// TIA Portal V20 export
// export: Created 2025-12-01T14:57:01.9840998Z, ExportSetting None, DisplayName Totally Integrated Automation Portal, DisplayVersion V20 Update 3, DisplayName TIA Portal Openness, DisplayVersion V20 Update 3, DisplayName TIA Portal Version Control Interface, DisplayVersion V20 Update 3, DisplayName STEP 7 Professional, DisplayVersion V20 Update 3, DisplayName STEP 7 Safety, DisplayVersion V20 Update 2, DisplayName WinCC Basic/Comfort/Advanced, DisplayVersion V20 Update 3, DisplayName WinCC Professional, DisplayVersion V20 Update 3, DisplayName WinCC Unified, DisplayVersion V20 Update 3
FUNCTION "FC465_Elevador_Continuo_Building" : Void   // FC465, LAD
TITLE = ELEVADOR CONTINUO
{ S7_Optimized_Access := 'FALSE' }
VERSION : 1.0
// Control para un elevador continuo con una única entrada y una única salida. si requiere de más salidas es necesario aplicar otro control para el movimiento y para el transportador abatible
// stored: AutoNumber false, SetENOAutomatically false
   VAR_INPUT
      NumeroMesa : UInt;
      NumeroMesaEntrada : UInt;
      NumeroMesaSalida : UInt;
      Termico_TEnt : Bool;
      Termico_TSal : Bool;
      Termico_Elev : Bool;
      pHs_Ent : Bool;
      Prot_Ent : Bool;
      pHs_Sal : Bool;
      Prot_Sal : Bool;
      Det_Sincr_Entrada : Bool;
      Det_Salida_Paro : Bool;
      Det_Salida_Emerg : Bool;
      AVTF_Ant : Bool;
      PTF_Sig : Bool;
      V_Permiso_Entrada : UDInt;
      V_Presencia_Entrada : UDInt;
      V_Paro_Elev : UDInt;
      V_Paro_Sal_ms : UDInt;
   END_VAR
   VAR_IN_OUT
      MAux_FP_Sincr : Bool;
      MAux_FN_Entrada : Bool;
      MAux_FP_Salida : Bool;
      Mem_TmpParoSal : Bool;
      Mem_Paro_Elev : Bool;
      out_Elevacion : Bool;
      out_Avance_Ent : Bool;
      out_Avance_Sal : Bool;
      out_AVTF_Sig : Bool;
      out_Carga_OK_Ant : Bool;
      Mem_TmpPermEntrada : Bool;
      Mem_TmpCentradoEntrada : Bool;
      Mem_TmpParoElev : Bool;
   END_VAR
   VAR_TEMP   // added for the SCL form of the ladder/FBD networks
      _w1 : Bool;
      _w2 : Bool;
   END_VAR
BEGIN

REGION Network 1: Marca General Error
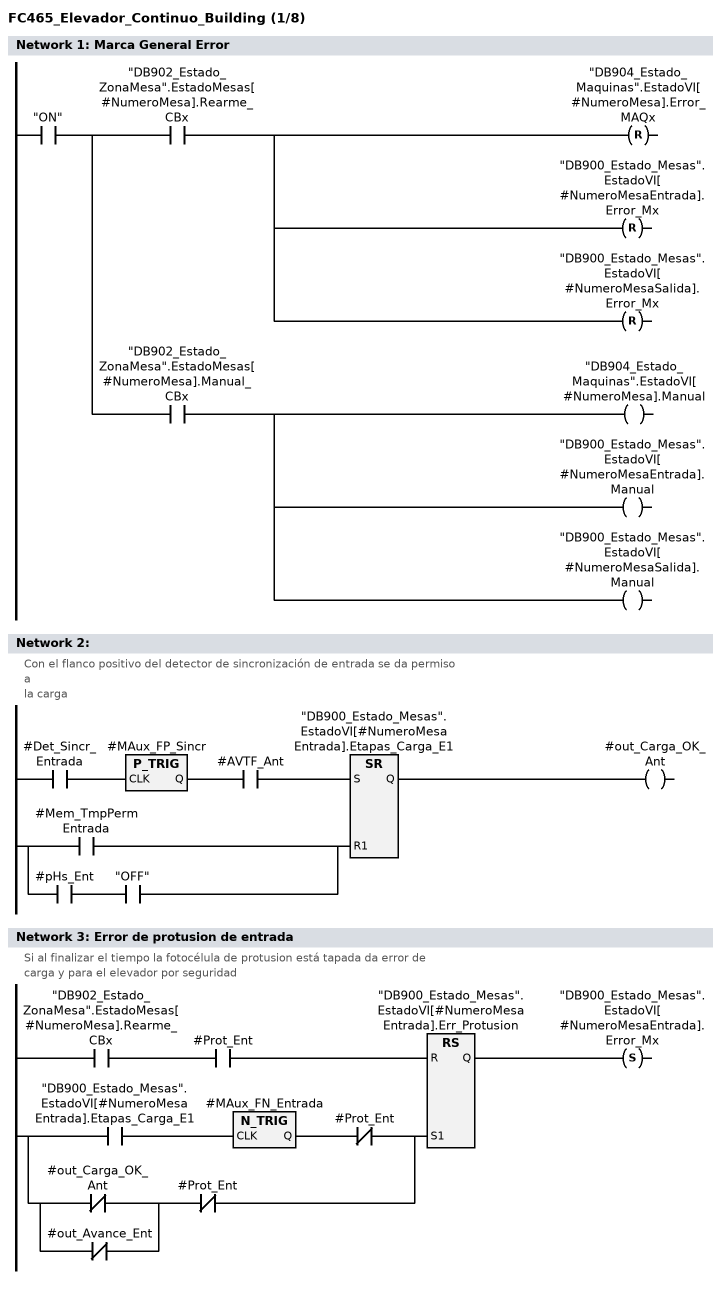
   RUNG wire#powerrail
      Contact( "ON" )
      wire#w1
      Contact( "DB902_Estado_ZonaMesa".EstadoMesas[#NumeroMesa].Rearme_CBx )
      wire#w2
      R_Coil( "DB904_Estado_Maquinas".EstadoVI[#NumeroMesa].Error_MAQx )
   END_RUNG
   RUNG wire#w2
      R_Coil( "DB900_Estado_Mesas".EstadoVI[#NumeroMesaEntrada].Error_Mx )
   END_RUNG
   RUNG wire#w2
      R_Coil( "DB900_Estado_Mesas".EstadoVI[#NumeroMesaSalida].Error_Mx )
   END_RUNG
   RUNG wire#w1
      Contact( "DB902_Estado_ZonaMesa".EstadoMesas[#NumeroMesa].Manual_CBx )
      wire#w3
      Coil( "DB904_Estado_Maquinas".EstadoVI[#NumeroMesa].Manual )
   END_RUNG
   RUNG wire#w3
      Coil( "DB900_Estado_Mesas".EstadoVI[#NumeroMesaEntrada].Manual )
   END_RUNG
   RUNG wire#w3
      Coil( "DB900_Estado_Mesas".EstadoVI[#NumeroMesaSalida].Manual )
   END_RUNG
   // the same network as SCL:
   #_w1 := "ON" AND "DB902_Estado_ZonaMesa".EstadoMesas[#NumeroMesa].Rearme_CBx;
   IF #_w1 THEN
       "DB904_Estado_Maquinas".EstadoVI[#NumeroMesa].Error_MAQx := FALSE;
       "DB900_Estado_Mesas".EstadoVI[#NumeroMesaEntrada].Error_Mx := FALSE;
       "DB900_Estado_Mesas".EstadoVI[#NumeroMesaSalida].Error_Mx := FALSE;
   END_IF;
   #_w2 := "ON" AND "DB902_Estado_ZonaMesa".EstadoMesas[#NumeroMesa].Manual_CBx;
   "DB904_Estado_Maquinas".EstadoVI[#NumeroMesa].Manual := "ON" AND "DB902_Estado_ZonaMesa".EstadoMesas[#NumeroMesa].Manual_CBx;
   "DB900_Estado_Mesas".EstadoVI[#NumeroMesaEntrada].Manual := #_w2;
   "DB900_Estado_Mesas".EstadoVI[#NumeroMesaSalida].Manual := #_w2;
END_REGION

REGION Network 2
   // Con el flanco positivo del detector de sincronización de entrada se da permiso 
   // a 
   // la carga
   RUNG wire#powerrail
      Contact( #Det_Sincr_Entrada )
      P_Trig( #MAux_FP_Sincr )
      Contact( #AVTF_Ant )
      S_SR(operand := "DB900_Estado_Mesas".EstadoVI[#NumeroMesaEntrada].Etapas_Carga_E1, r1 := wire#w1)
      Coil( #out_Carga_OK_Ant )
   END_RUNG
   RUNG wire#powerrail
      Contact( #Mem_TmpPermEntrada )
   END_RUNG wire#w1
   RUNG wire#powerrail
      Contact( #pHs_Ent )
      Contact( "OFF" )
   END_RUNG wire#w1
   // the same network as SCL:
   #_w1 := #Det_Sincr_Entrada AND NOT #MAux_FP_Sincr;   // rising edge
   #MAux_FP_Sincr := #Det_Sincr_Entrada;
   IF #_w1 AND #AVTF_Ant THEN
       "DB900_Estado_Mesas".EstadoVI[#NumeroMesaEntrada].Etapas_Carga_E1 := TRUE;   // SR flip-flop
   END_IF;
   IF #Mem_TmpPermEntrada OR (#pHs_Ent AND "OFF") THEN
       "DB900_Estado_Mesas".EstadoVI[#NumeroMesaEntrada].Etapas_Carga_E1 := FALSE;
   END_IF;
   #out_Carga_OK_Ant := "DB900_Estado_Mesas".EstadoVI[#NumeroMesaEntrada].Etapas_Carga_E1;
END_REGION

REGION Network 3: Error de protusion de entrada
   // Si al finalizar el tiempo la fotocélula de protusion está tapada da error de 
   // carga y para el elevador por seguridad
   RUNG wire#powerrail
      Contact( "DB902_Estado_ZonaMesa".EstadoMesas[#NumeroMesa].Rearme_CBx )
      Contact( #Prot_Ent )
      S_RS(operand := "DB900_Estado_Mesas".EstadoVI[#NumeroMesaEntrada].Err_Protusion, s1 := wire#w2)
      S_Coil( "DB900_Estado_Mesas".EstadoVI[#NumeroMesaEntrada].Error_Mx )
   END_RUNG
   RUNG wire#powerrail
      Contact( "DB900_Estado_Mesas".EstadoVI[#NumeroMesaEntrada].Etapas_Carga_E1 )
      N_Trig( #MAux_FN_Entrada )
      I_Contact( #Prot_Ent )
   END_RUNG wire#w2
   RUNG wire#powerrail
      I_Contact( #out_Carga_OK_Ant )
      wire#w1
      I_Contact( #Prot_Ent )
   END_RUNG wire#w2
   RUNG wire#powerrail
      I_Contact( #out_Avance_Ent )
   END_RUNG wire#w1
   // the same network as SCL:
   #_w1 := NOT "DB900_Estado_Mesas".EstadoVI[#NumeroMesaEntrada].Etapas_Carga_E1 AND #MAux_FN_Entrada;   // falling edge
   #MAux_FN_Entrada := "DB900_Estado_Mesas".EstadoVI[#NumeroMesaEntrada].Etapas_Carga_E1;
   IF "DB902_Estado_ZonaMesa".EstadoMesas[#NumeroMesa].Rearme_CBx AND #Prot_Ent THEN
       "DB900_Estado_Mesas".EstadoVI[#NumeroMesaEntrada].Err_Protusion := FALSE;   // RS flip-flop
   END_IF;
   IF (#_w1 AND NOT #Prot_Ent) OR ((NOT #out_Carga_OK_Ant OR NOT #out_Avance_Ent) AND NOT #Prot_Ent) THEN
       "DB900_Estado_Mesas".EstadoVI[#NumeroMesaEntrada].Err_Protusion := TRUE;
   END_IF;
   IF "DB900_Estado_Mesas".EstadoVI[#NumeroMesaEntrada].Err_Protusion THEN
       "DB900_Estado_Mesas".EstadoVI[#NumeroMesaEntrada].Error_Mx := TRUE;
   END_IF;
END_REGION

REGION Network 4: Error protusion de salida
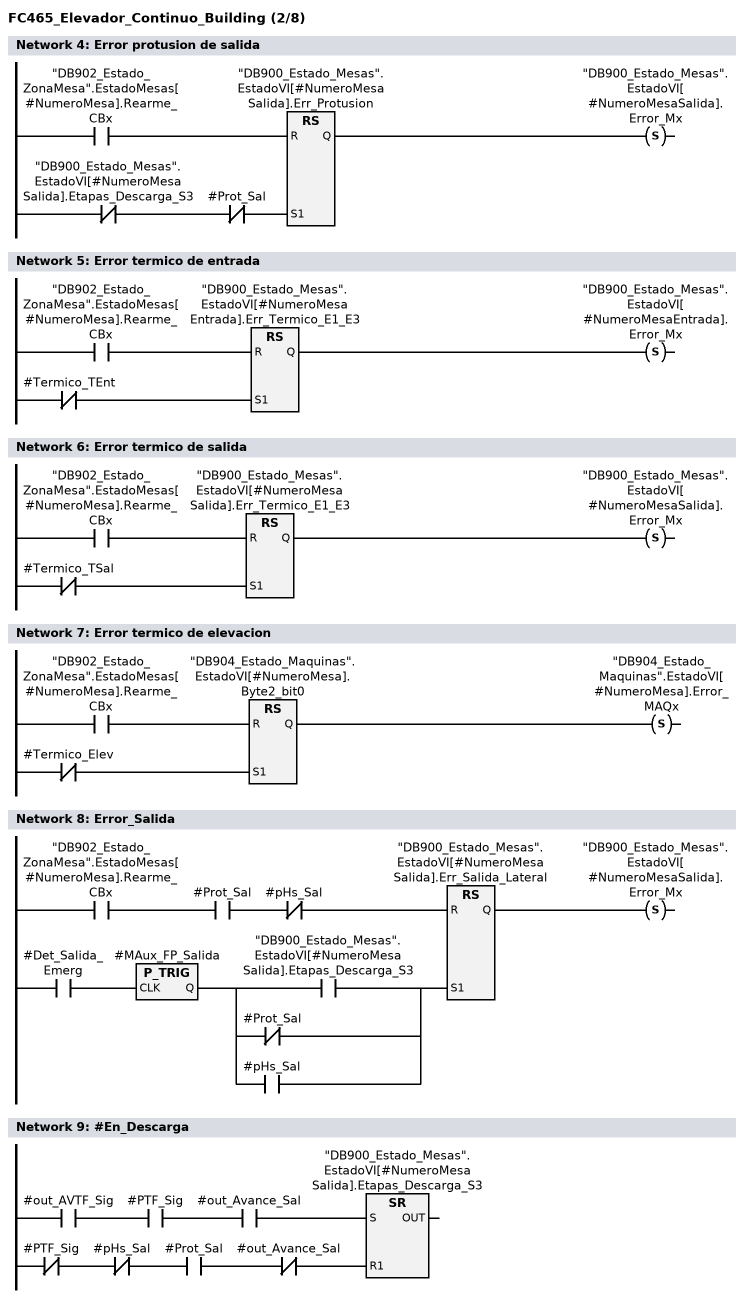
   RUNG wire#powerrail
      Contact( "DB902_Estado_ZonaMesa".EstadoMesas[#NumeroMesa].Rearme_CBx )
      S_RS(operand := "DB900_Estado_Mesas".EstadoVI[#NumeroMesaSalida].Err_Protusion, s1 := wire#w1)
      S_Coil( "DB900_Estado_Mesas".EstadoVI[#NumeroMesaSalida].Error_Mx )
   END_RUNG
   RUNG wire#powerrail
      I_Contact( "DB900_Estado_Mesas".EstadoVI[#NumeroMesaSalida].Etapas_Descarga_S3 )
      I_Contact( #Prot_Sal )
   END_RUNG wire#w1
   // the same network as SCL:
   #_w1 := NOT "DB900_Estado_Mesas".EstadoVI[#NumeroMesaSalida].Etapas_Descarga_S3 AND NOT #Prot_Sal;
   IF "DB902_Estado_ZonaMesa".EstadoMesas[#NumeroMesa].Rearme_CBx THEN
       "DB900_Estado_Mesas".EstadoVI[#NumeroMesaSalida].Err_Protusion := FALSE;   // RS flip-flop
   END_IF;
   IF #_w1 THEN "DB900_Estado_Mesas".EstadoVI[#NumeroMesaSalida].Err_Protusion := TRUE; END_IF;
   IF "DB900_Estado_Mesas".EstadoVI[#NumeroMesaSalida].Err_Protusion THEN
       "DB900_Estado_Mesas".EstadoVI[#NumeroMesaSalida].Error_Mx := TRUE;
   END_IF;
END_REGION

REGION Network 5: Error termico de entrada
   RUNG wire#powerrail
      Contact( "DB902_Estado_ZonaMesa".EstadoMesas[#NumeroMesa].Rearme_CBx )
      S_RS(operand := "DB900_Estado_Mesas".EstadoVI[#NumeroMesaEntrada].Err_Termico_E1_E3, s1 := wire#w1)
      S_Coil( "DB900_Estado_Mesas".EstadoVI[#NumeroMesaEntrada].Error_Mx )
   END_RUNG
   RUNG wire#powerrail
      I_Contact( #Termico_TEnt )
   END_RUNG wire#w1
   // the same network as SCL:
   IF "DB902_Estado_ZonaMesa".EstadoMesas[#NumeroMesa].Rearme_CBx THEN
       "DB900_Estado_Mesas".EstadoVI[#NumeroMesaEntrada].Err_Termico_E1_E3 := FALSE;   // RS flip-flop
   END_IF;
   IF NOT #Termico_TEnt THEN
       "DB900_Estado_Mesas".EstadoVI[#NumeroMesaEntrada].Err_Termico_E1_E3 := TRUE;
   END_IF;
   IF "DB900_Estado_Mesas".EstadoVI[#NumeroMesaEntrada].Err_Termico_E1_E3 THEN
       "DB900_Estado_Mesas".EstadoVI[#NumeroMesaEntrada].Error_Mx := TRUE;
   END_IF;
END_REGION

REGION Network 6: Error termico de salida
   RUNG wire#powerrail
      Contact( "DB902_Estado_ZonaMesa".EstadoMesas[#NumeroMesa].Rearme_CBx )
      S_RS(operand := "DB900_Estado_Mesas".EstadoVI[#NumeroMesaSalida].Err_Termico_E1_E3, s1 := wire#w1)
      S_Coil( "DB900_Estado_Mesas".EstadoVI[#NumeroMesaSalida].Error_Mx )
   END_RUNG
   RUNG wire#powerrail
      I_Contact( #Termico_TSal )
   END_RUNG wire#w1
   // the same network as SCL:
   IF "DB902_Estado_ZonaMesa".EstadoMesas[#NumeroMesa].Rearme_CBx THEN
       "DB900_Estado_Mesas".EstadoVI[#NumeroMesaSalida].Err_Termico_E1_E3 := FALSE;   // RS flip-flop
   END_IF;
   IF NOT #Termico_TSal THEN
       "DB900_Estado_Mesas".EstadoVI[#NumeroMesaSalida].Err_Termico_E1_E3 := TRUE;
   END_IF;
   IF "DB900_Estado_Mesas".EstadoVI[#NumeroMesaSalida].Err_Termico_E1_E3 THEN
       "DB900_Estado_Mesas".EstadoVI[#NumeroMesaSalida].Error_Mx := TRUE;
   END_IF;
END_REGION

REGION Network 7: Error termico de elevacion
   RUNG wire#powerrail
      Contact( "DB902_Estado_ZonaMesa".EstadoMesas[#NumeroMesa].Rearme_CBx )
      S_RS(operand := "DB904_Estado_Maquinas".EstadoVI[#NumeroMesa].Byte2_bit0, s1 := wire#w1)
      S_Coil( "DB904_Estado_Maquinas".EstadoVI[#NumeroMesa].Error_MAQx )
   END_RUNG
   RUNG wire#powerrail
      I_Contact( #Termico_Elev )
   END_RUNG wire#w1
   // the same network as SCL:
   IF "DB902_Estado_ZonaMesa".EstadoMesas[#NumeroMesa].Rearme_CBx THEN
       "DB904_Estado_Maquinas".EstadoVI[#NumeroMesa].Byte2_bit0 := FALSE;   // RS flip-flop
   END_IF;
   IF NOT #Termico_Elev THEN "DB904_Estado_Maquinas".EstadoVI[#NumeroMesa].Byte2_bit0 := TRUE; END_IF;
   IF "DB904_Estado_Maquinas".EstadoVI[#NumeroMesa].Byte2_bit0 THEN
       "DB904_Estado_Maquinas".EstadoVI[#NumeroMesa].Error_MAQx := TRUE;
   END_IF;
END_REGION

REGION Network 8: Error_Salida
   RUNG wire#powerrail
      Contact( "DB902_Estado_ZonaMesa".EstadoMesas[#NumeroMesa].Rearme_CBx )
      Contact( #Prot_Sal )
      I_Contact( #pHs_Sal )
      S_RS(operand := "DB900_Estado_Mesas".EstadoVI[#NumeroMesaSalida].Err_Salida_Lateral, s1 := wire#w2)
      S_Coil( "DB900_Estado_Mesas".EstadoVI[#NumeroMesaSalida].Error_Mx )
   END_RUNG
   RUNG wire#powerrail
      Contact( #Det_Salida_Emerg )
      P_Trig( #MAux_FP_Salida )
      wire#w1
      Contact( "DB900_Estado_Mesas".EstadoVI[#NumeroMesaSalida].Etapas_Descarga_S3 )
   END_RUNG wire#w2
   RUNG wire#w1
      I_Contact( #Prot_Sal )
   END_RUNG wire#w2
   RUNG wire#w1
      Contact( #pHs_Sal )
   END_RUNG wire#w2
   // the same network as SCL:
   #_w1 := #Det_Salida_Emerg AND NOT #MAux_FP_Salida;   // rising edge
   #MAux_FP_Salida := #Det_Salida_Emerg;
   #_w2 := #_w1 AND ("DB900_Estado_Mesas".EstadoVI[#NumeroMesaSalida].Etapas_Descarga_S3 OR NOT #Prot_Sal OR #pHs_Sal);
   IF "DB902_Estado_ZonaMesa".EstadoMesas[#NumeroMesa].Rearme_CBx AND #Prot_Sal AND NOT #pHs_Sal THEN
       "DB900_Estado_Mesas".EstadoVI[#NumeroMesaSalida].Err_Salida_Lateral := FALSE;   // RS flip-flop
   END_IF;
   IF #_w2 THEN "DB900_Estado_Mesas".EstadoVI[#NumeroMesaSalida].Err_Salida_Lateral := TRUE; END_IF;
   IF "DB900_Estado_Mesas".EstadoVI[#NumeroMesaSalida].Err_Salida_Lateral THEN
       "DB900_Estado_Mesas".EstadoVI[#NumeroMesaSalida].Error_Mx := TRUE;
   END_IF;
END_REGION

REGION Network 9: #En_Descarga
   RUNG wire#powerrail
      Contact( #out_AVTF_Sig )
      Contact( #PTF_Sig )
      Contact( #out_Avance_Sal )
      S_SR(operand := "DB900_Estado_Mesas".EstadoVI[#NumeroMesaSalida].Etapas_Descarga_S3, r1 := wire#w1)
   END_RUNG
   RUNG wire#powerrail
      I_Contact( #PTF_Sig )
      I_Contact( #pHs_Sal )
      Contact( #Prot_Sal )
      I_Contact( #out_Avance_Sal )
   END_RUNG wire#w1
   // the same network as SCL:
   IF #out_AVTF_Sig AND #PTF_Sig AND #out_Avance_Sal THEN
       "DB900_Estado_Mesas".EstadoVI[#NumeroMesaSalida].Etapas_Descarga_S3 := TRUE;   // SR flip-flop
   END_IF;
   IF NOT #PTF_Sig AND NOT #pHs_Sal AND #Prot_Sal AND NOT #out_Avance_Sal THEN
       "DB900_Estado_Mesas".EstadoVI[#NumeroMesaSalida].Etapas_Descarga_S3 := FALSE;
   END_IF;
END_REGION

REGION Network 10: Paro elevador por estar ocupada la salida
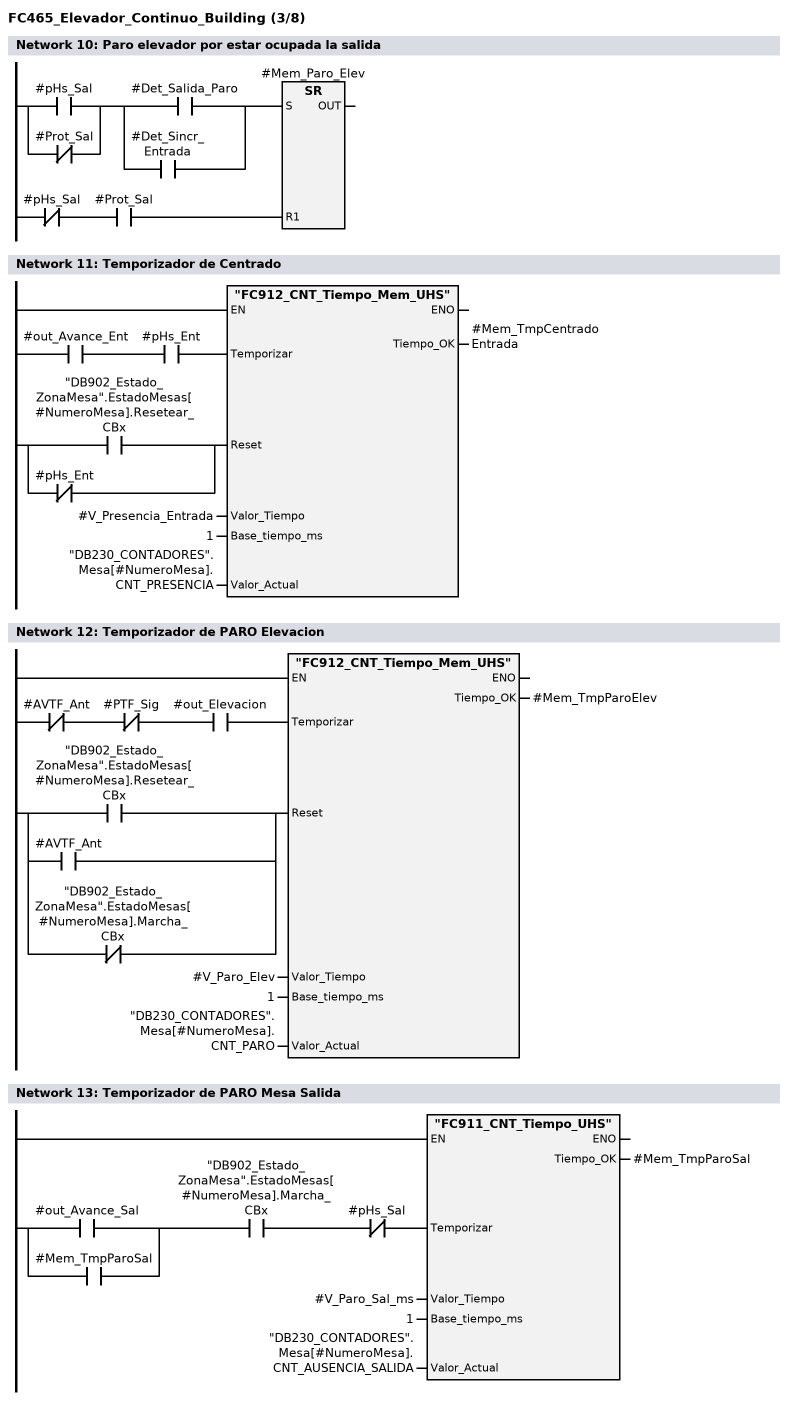
   RUNG wire#powerrail
      Contact( #pHs_Sal )
      wire#w1
      Contact( #Det_Salida_Paro )
      wire#w2
      S_SR(operand := #Mem_Paro_Elev, r1 := wire#w3)
   END_RUNG
   RUNG wire#powerrail
      I_Contact( #Prot_Sal )
   END_RUNG wire#w1
   RUNG wire#w1
      Contact( #Det_Sincr_Entrada )
   END_RUNG wire#w2
   RUNG wire#powerrail
      I_Contact( #pHs_Sal )
      Contact( #Prot_Sal )
   END_RUNG wire#w3
   // the same network as SCL:
   IF (#pHs_Sal OR NOT #Prot_Sal) AND (#Det_Salida_Paro OR #Det_Sincr_Entrada) THEN
       #Mem_Paro_Elev := TRUE;   // SR flip-flop
   END_IF;
   IF NOT #pHs_Sal AND #Prot_Sal THEN #Mem_Paro_Elev := FALSE; END_IF;
END_REGION

REGION Network 11: Temporizador de Centrado
   RUNG wire#powerrail
      "FC912_CNT_Tiempo_Mem_UHS"(Temporizar := wire#w1, Reset := wire#w2, Valor_Tiempo := #V_Presencia_Entrada, Base_tiempo_ms := 1, Valor_Actual := "DB230_CONTADORES".Mesa[#NumeroMesa].CNT_PRESENCIA, Tiempo_OK => #Mem_TmpCentradoEntrada)
   END_RUNG
   RUNG wire#powerrail
      Contact( #out_Avance_Ent )
      Contact( #pHs_Ent )
   END_RUNG wire#w1
   RUNG wire#powerrail
      Contact( "DB902_Estado_ZonaMesa".EstadoMesas[#NumeroMesa].Resetear_CBx )
   END_RUNG wire#w2
   RUNG wire#powerrail
      I_Contact( #pHs_Ent )
   END_RUNG wire#w2
   // the same network as SCL:
   "FC912_CNT_Tiempo_Mem_UHS"(Temporizar := #out_Avance_Ent AND #pHs_Ent,
                           Reset := "DB902_Estado_ZonaMesa".EstadoMesas[#NumeroMesa].Resetear_CBx OR NOT #pHs_Ent,
                           Valor_Tiempo := #V_Presencia_Entrada,
                           Base_tiempo_ms := 1,
                           Valor_Actual := "DB230_CONTADORES".Mesa[#NumeroMesa].CNT_PRESENCIA,
                           Tiempo_OK => #Mem_TmpCentradoEntrada);
END_REGION

REGION Network 12: Temporizador de PARO Elevacion
   RUNG wire#powerrail
      "FC912_CNT_Tiempo_Mem_UHS"(Temporizar := wire#w1, Reset := wire#w2, Valor_Tiempo := #V_Paro_Elev, Base_tiempo_ms := 1, Valor_Actual := "DB230_CONTADORES".Mesa[#NumeroMesa].CNT_PARO, Tiempo_OK => #Mem_TmpParoElev)
   END_RUNG
   RUNG wire#powerrail
      I_Contact( #AVTF_Ant )
      I_Contact( #PTF_Sig )
      Contact( #out_Elevacion )
   END_RUNG wire#w1
   RUNG wire#powerrail
      Contact( "DB902_Estado_ZonaMesa".EstadoMesas[#NumeroMesa].Resetear_CBx )
   END_RUNG wire#w2
   RUNG wire#powerrail
      Contact( #AVTF_Ant )
   END_RUNG wire#w2
   RUNG wire#powerrail
      I_Contact( "DB902_Estado_ZonaMesa".EstadoMesas[#NumeroMesa].Marcha_CBx )
   END_RUNG wire#w2
   // the same network as SCL:
   "FC912_CNT_Tiempo_Mem_UHS"(Temporizar := NOT #AVTF_Ant AND NOT #PTF_Sig AND #out_Elevacion,
                           Reset := "DB902_Estado_ZonaMesa".EstadoMesas[#NumeroMesa].Resetear_CBx OR #AVTF_Ant OR NOT "DB902_Estado_ZonaMesa".EstadoMesas[#NumeroMesa].Marcha_CBx,
                           Valor_Tiempo := #V_Paro_Elev,
                           Base_tiempo_ms := 1,
                           Valor_Actual := "DB230_CONTADORES".Mesa[#NumeroMesa].CNT_PARO,
                           Tiempo_OK => #Mem_TmpParoElev);
END_REGION

REGION Network 13: Temporizador de PARO Mesa Salida
   RUNG wire#powerrail
      "FC911_CNT_Tiempo_UHS"(Temporizar := wire#w2, Valor_Tiempo := #V_Paro_Sal_ms, Base_tiempo_ms := 1, Valor_Actual := "DB230_CONTADORES".Mesa[#NumeroMesa].CNT_AUSENCIA_SALIDA, Tiempo_OK => #Mem_TmpParoSal)
   END_RUNG
   RUNG wire#powerrail
      Contact( #out_Avance_Sal )
      wire#w1
      Contact( "DB902_Estado_ZonaMesa".EstadoMesas[#NumeroMesa].Marcha_CBx )
      I_Contact( #pHs_Sal )
   END_RUNG wire#w2
   RUNG wire#powerrail
      Contact( #Mem_TmpParoSal )
   END_RUNG wire#w1
   // the same network as SCL:
   "FC911_CNT_Tiempo_UHS"(Temporizar := (#out_Avance_Sal OR #Mem_TmpParoSal) AND "DB902_Estado_ZonaMesa".EstadoMesas[#NumeroMesa].Marcha_CBx AND NOT #pHs_Sal,
                          Valor_Tiempo := #V_Paro_Sal_ms,
                          Base_tiempo_ms := 1,
                          Valor_Actual := "DB230_CONTADORES".Mesa[#NumeroMesa].CNT_AUSENCIA_SALIDA,
                          Tiempo_OK => #Mem_TmpParoSal);
END_REGION

REGION Network 14: Temporizador de PARO E2
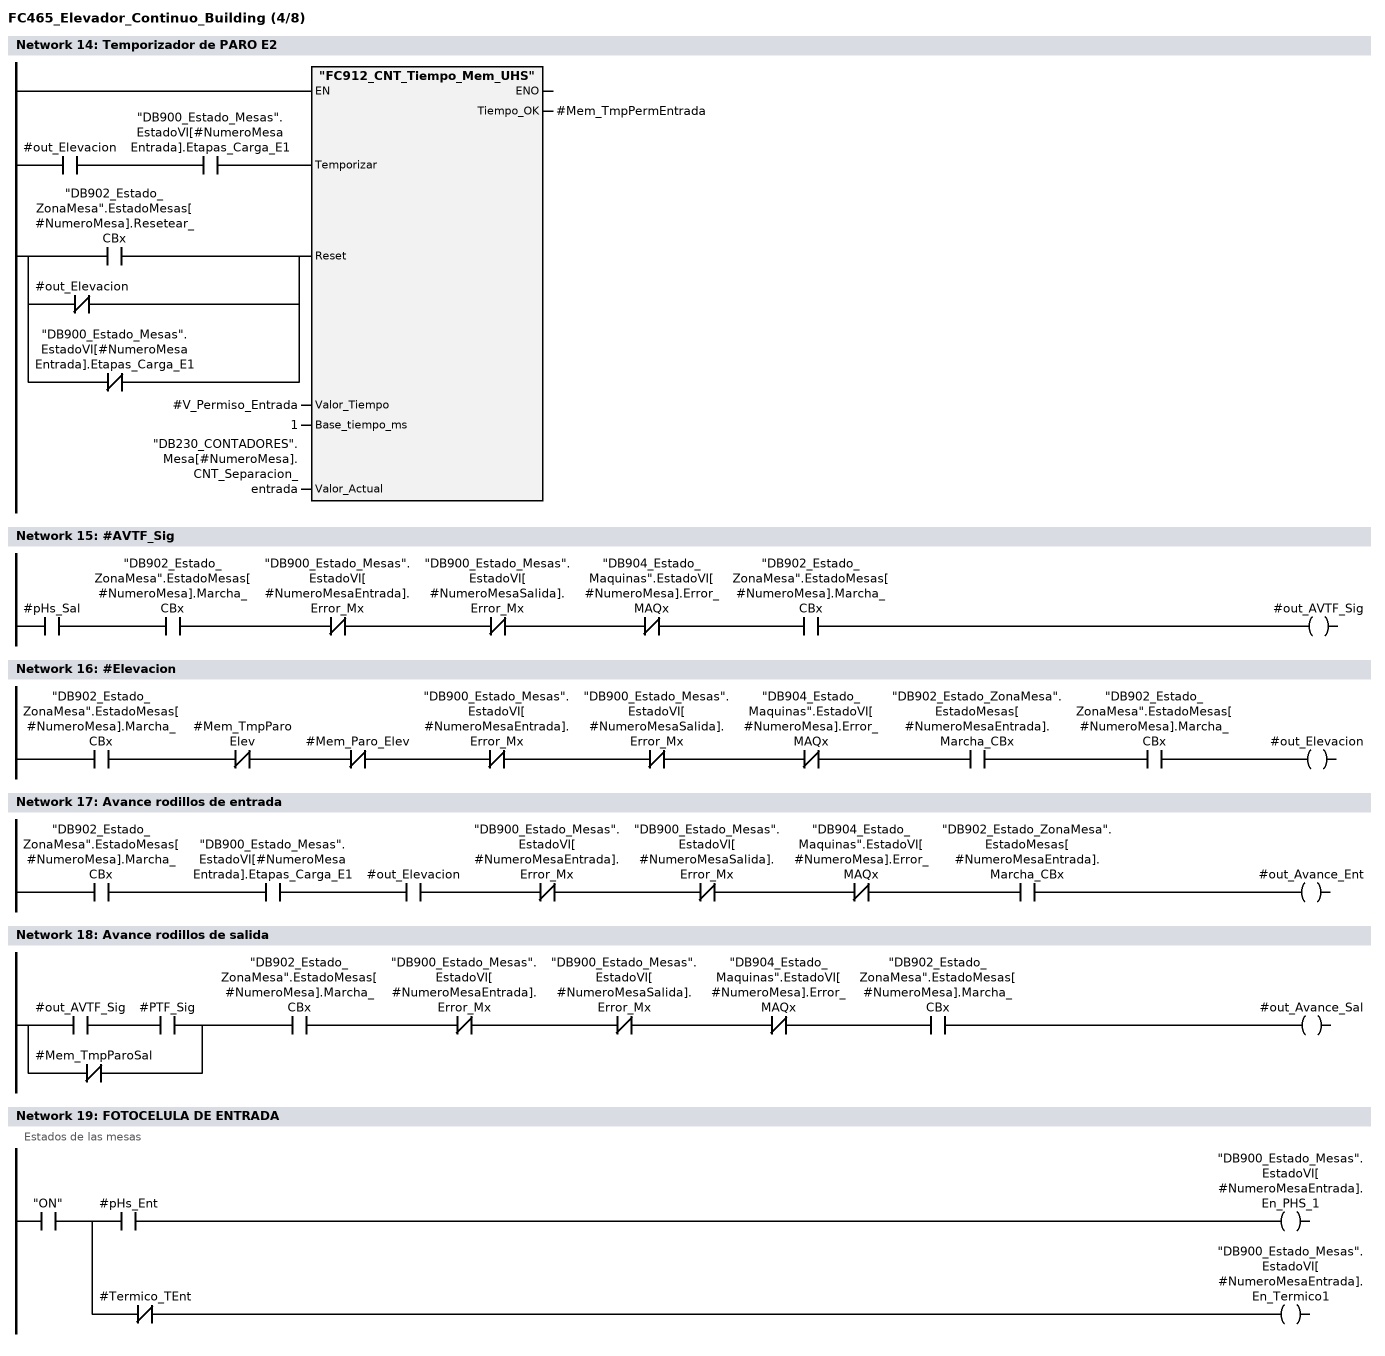
   RUNG wire#powerrail
      "FC912_CNT_Tiempo_Mem_UHS"(Temporizar := wire#w1, Reset := wire#w2, Valor_Tiempo := #V_Permiso_Entrada, Base_tiempo_ms := 1, Valor_Actual := "DB230_CONTADORES".Mesa[#NumeroMesa].CNT_Separacion_entrada, Tiempo_OK => #Mem_TmpPermEntrada)
   END_RUNG
   RUNG wire#powerrail
      Contact( #out_Elevacion )
      Contact( "DB900_Estado_Mesas".EstadoVI[#NumeroMesaEntrada].Etapas_Carga_E1 )
   END_RUNG wire#w1
   RUNG wire#powerrail
      Contact( "DB902_Estado_ZonaMesa".EstadoMesas[#NumeroMesa].Resetear_CBx )
   END_RUNG wire#w2
   RUNG wire#powerrail
      I_Contact( #out_Elevacion )
   END_RUNG wire#w2
   RUNG wire#powerrail
      I_Contact( "DB900_Estado_Mesas".EstadoVI[#NumeroMesaEntrada].Etapas_Carga_E1 )
   END_RUNG wire#w2
   // the same network as SCL:
   "FC912_CNT_Tiempo_Mem_UHS"(Temporizar := #out_Elevacion AND "DB900_Estado_Mesas".EstadoVI[#NumeroMesaEntrada].Etapas_Carga_E1,
                           Reset := "DB902_Estado_ZonaMesa".EstadoMesas[#NumeroMesa].Resetear_CBx OR NOT #out_Elevacion OR NOT "DB900_Estado_Mesas".EstadoVI[#NumeroMesaEntrada].Etapas_Carga_E1,
                           Valor_Tiempo := #V_Permiso_Entrada,
                           Base_tiempo_ms := 1,
                           Valor_Actual := "DB230_CONTADORES".Mesa[#NumeroMesa].CNT_Separacion_entrada,
                           Tiempo_OK => #Mem_TmpPermEntrada);
END_REGION

REGION Network 15: #AVTF_Sig
   RUNG wire#powerrail
      Contact( #pHs_Sal )
      Contact( "DB902_Estado_ZonaMesa".EstadoMesas[#NumeroMesa].Marcha_CBx )
      I_Contact( "DB900_Estado_Mesas".EstadoVI[#NumeroMesaEntrada].Error_Mx )
      I_Contact( "DB900_Estado_Mesas".EstadoVI[#NumeroMesaSalida].Error_Mx )
      I_Contact( "DB904_Estado_Maquinas".EstadoVI[#NumeroMesa].Error_MAQx )
      Contact( "DB902_Estado_ZonaMesa".EstadoMesas[#NumeroMesa].Marcha_CBx )
      Coil( #out_AVTF_Sig )
   END_RUNG
   // the same network as SCL:
   #out_AVTF_Sig := #pHs_Sal AND "DB902_Estado_ZonaMesa".EstadoMesas[#NumeroMesa].Marcha_CBx AND NOT "DB900_Estado_Mesas".EstadoVI[#NumeroMesaEntrada].Error_Mx AND NOT "DB900_Estado_Mesas".EstadoVI[#NumeroMesaSalida].Error_Mx AND NOT "DB904_Estado_Maquinas".EstadoVI[#NumeroMesa].Error_MAQx AND "DB902_Estado_ZonaMesa".EstadoMesas[#NumeroMesa].Marcha_CBx;
END_REGION

REGION Network 16: #Elevacion
   RUNG wire#powerrail
      Contact( "DB902_Estado_ZonaMesa".EstadoMesas[#NumeroMesa].Marcha_CBx )
      I_Contact( #Mem_TmpParoElev )
      I_Contact( #Mem_Paro_Elev )
      I_Contact( "DB900_Estado_Mesas".EstadoVI[#NumeroMesaEntrada].Error_Mx )
      I_Contact( "DB900_Estado_Mesas".EstadoVI[#NumeroMesaSalida].Error_Mx )
      I_Contact( "DB904_Estado_Maquinas".EstadoVI[#NumeroMesa].Error_MAQx )
      Contact( "DB902_Estado_ZonaMesa".EstadoMesas[#NumeroMesaEntrada].Marcha_CBx )
      Contact( "DB902_Estado_ZonaMesa".EstadoMesas[#NumeroMesa].Marcha_CBx )
      Coil( #out_Elevacion )
   END_RUNG
   // the same network as SCL:
   #out_Elevacion := "DB902_Estado_ZonaMesa".EstadoMesas[#NumeroMesa].Marcha_CBx AND NOT #Mem_TmpParoElev AND NOT #Mem_Paro_Elev AND NOT "DB900_Estado_Mesas".EstadoVI[#NumeroMesaEntrada].Error_Mx AND NOT "DB900_Estado_Mesas".EstadoVI[#NumeroMesaSalida].Error_Mx AND NOT "DB904_Estado_Maquinas".EstadoVI[#NumeroMesa].Error_MAQx AND "DB902_Estado_ZonaMesa".EstadoMesas[#NumeroMesaEntrada].Marcha_CBx AND "DB902_Estado_ZonaMesa".EstadoMesas[#NumeroMesa].Marcha_CBx;
END_REGION

REGION Network 17: Avance rodillos de entrada
   RUNG wire#powerrail
      Contact( "DB902_Estado_ZonaMesa".EstadoMesas[#NumeroMesa].Marcha_CBx )
      Contact( "DB900_Estado_Mesas".EstadoVI[#NumeroMesaEntrada].Etapas_Carga_E1 )
      Contact( #out_Elevacion )
      I_Contact( "DB900_Estado_Mesas".EstadoVI[#NumeroMesaEntrada].Error_Mx )
      I_Contact( "DB900_Estado_Mesas".EstadoVI[#NumeroMesaSalida].Error_Mx )
      I_Contact( "DB904_Estado_Maquinas".EstadoVI[#NumeroMesa].Error_MAQx )
      Contact( "DB902_Estado_ZonaMesa".EstadoMesas[#NumeroMesaEntrada].Marcha_CBx )
      Coil( #out_Avance_Ent )
   END_RUNG
   // the same network as SCL:
   #out_Avance_Ent := "DB902_Estado_ZonaMesa".EstadoMesas[#NumeroMesa].Marcha_CBx AND "DB900_Estado_Mesas".EstadoVI[#NumeroMesaEntrada].Etapas_Carga_E1 AND #out_Elevacion AND NOT "DB900_Estado_Mesas".EstadoVI[#NumeroMesaEntrada].Error_Mx AND NOT "DB900_Estado_Mesas".EstadoVI[#NumeroMesaSalida].Error_Mx AND NOT "DB904_Estado_Maquinas".EstadoVI[#NumeroMesa].Error_MAQx AND "DB902_Estado_ZonaMesa".EstadoMesas[#NumeroMesaEntrada].Marcha_CBx;
END_REGION

REGION Network 18: Avance rodillos de salida
   RUNG wire#powerrail
      Contact( #out_AVTF_Sig )
      Contact( #PTF_Sig )
      wire#w1
      Contact( "DB902_Estado_ZonaMesa".EstadoMesas[#NumeroMesa].Marcha_CBx )
      I_Contact( "DB900_Estado_Mesas".EstadoVI[#NumeroMesaEntrada].Error_Mx )
      I_Contact( "DB900_Estado_Mesas".EstadoVI[#NumeroMesaSalida].Error_Mx )
      I_Contact( "DB904_Estado_Maquinas".EstadoVI[#NumeroMesa].Error_MAQx )
      Contact( "DB902_Estado_ZonaMesa".EstadoMesas[#NumeroMesa].Marcha_CBx )
      Coil( #out_Avance_Sal )
   END_RUNG
   RUNG wire#powerrail
      I_Contact( #Mem_TmpParoSal )
   END_RUNG wire#w1
   // the same network as SCL:
   #out_Avance_Sal := ((#out_AVTF_Sig AND #PTF_Sig) OR NOT #Mem_TmpParoSal) AND "DB902_Estado_ZonaMesa".EstadoMesas[#NumeroMesa].Marcha_CBx AND NOT "DB900_Estado_Mesas".EstadoVI[#NumeroMesaEntrada].Error_Mx AND NOT "DB900_Estado_Mesas".EstadoVI[#NumeroMesaSalida].Error_Mx AND NOT "DB904_Estado_Maquinas".EstadoVI[#NumeroMesa].Error_MAQx AND "DB902_Estado_ZonaMesa".EstadoMesas[#NumeroMesa].Marcha_CBx;
END_REGION

REGION Network 19: FOTOCELULA DE ENTRADA
   // Estados de las mesas
   RUNG wire#powerrail
      Contact( "ON" )
      wire#w1
      Contact( #pHs_Ent )
      Coil( "DB900_Estado_Mesas".EstadoVI[#NumeroMesaEntrada].En_PHS_1 )
   END_RUNG
   RUNG wire#w1
      I_Contact( #Termico_TEnt )
      Coil( "DB900_Estado_Mesas".EstadoVI[#NumeroMesaEntrada].En_Termico1 )
   END_RUNG
   // the same network as SCL:
   "DB900_Estado_Mesas".EstadoVI[#NumeroMesaEntrada].En_PHS_1 := "ON" AND #pHs_Ent;
   "DB900_Estado_Mesas".EstadoVI[#NumeroMesaEntrada].En_Termico1 := "ON" AND NOT #Termico_TEnt;
END_REGION

REGION Network 20: ESTADOS MESA ENTRADA
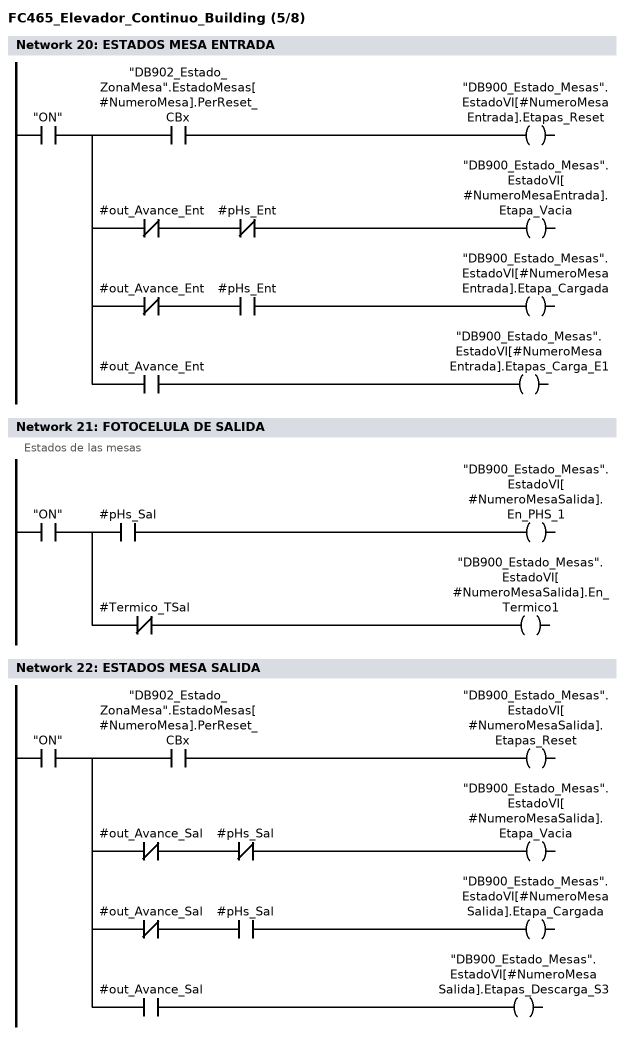
   RUNG wire#powerrail
      Contact( "ON" )
      wire#w1
      Contact( "DB902_Estado_ZonaMesa".EstadoMesas[#NumeroMesa].PerReset_CBx )
      Coil( "DB900_Estado_Mesas".EstadoVI[#NumeroMesaEntrada].Etapas_Reset )
   END_RUNG
   RUNG wire#w1
      I_Contact( #out_Avance_Ent )
      I_Contact( #pHs_Ent )
      Coil( "DB900_Estado_Mesas".EstadoVI[#NumeroMesaEntrada].Etapa_Vacia )
   END_RUNG
   RUNG wire#w1
      I_Contact( #out_Avance_Ent )
      Contact( #pHs_Ent )
      Coil( "DB900_Estado_Mesas".EstadoVI[#NumeroMesaEntrada].Etapa_Cargada )
   END_RUNG
   RUNG wire#w1
      Contact( #out_Avance_Ent )
      Coil( "DB900_Estado_Mesas".EstadoVI[#NumeroMesaEntrada].Etapas_Carga_E1 )
   END_RUNG
   // the same network as SCL:
   "DB900_Estado_Mesas".EstadoVI[#NumeroMesaEntrada].Etapas_Reset := "ON" AND "DB902_Estado_ZonaMesa".EstadoMesas[#NumeroMesa].PerReset_CBx;
   "DB900_Estado_Mesas".EstadoVI[#NumeroMesaEntrada].Etapa_Vacia := "ON" AND NOT #out_Avance_Ent AND NOT #pHs_Ent;
   "DB900_Estado_Mesas".EstadoVI[#NumeroMesaEntrada].Etapa_Cargada := "ON" AND NOT #out_Avance_Ent AND #pHs_Ent;
   "DB900_Estado_Mesas".EstadoVI[#NumeroMesaEntrada].Etapas_Carga_E1 := "ON" AND #out_Avance_Ent;
END_REGION

REGION Network 21: FOTOCELULA DE SALIDA
   // Estados de las mesas
   RUNG wire#powerrail
      Contact( "ON" )
      wire#w1
      Contact( #pHs_Sal )
      Coil( "DB900_Estado_Mesas".EstadoVI[#NumeroMesaSalida].En_PHS_1 )
   END_RUNG
   RUNG wire#w1
      I_Contact( #Termico_TSal )
      Coil( "DB900_Estado_Mesas".EstadoVI[#NumeroMesaSalida].En_Termico1 )
   END_RUNG
   // the same network as SCL:
   "DB900_Estado_Mesas".EstadoVI[#NumeroMesaSalida].En_PHS_1 := "ON" AND #pHs_Sal;
   "DB900_Estado_Mesas".EstadoVI[#NumeroMesaSalida].En_Termico1 := "ON" AND NOT #Termico_TSal;
END_REGION

REGION Network 22: ESTADOS MESA SALIDA
   RUNG wire#powerrail
      Contact( "ON" )
      wire#w1
      Contact( "DB902_Estado_ZonaMesa".EstadoMesas[#NumeroMesa].PerReset_CBx )
      Coil( "DB900_Estado_Mesas".EstadoVI[#NumeroMesaSalida].Etapas_Reset )
   END_RUNG
   RUNG wire#w1
      I_Contact( #out_Avance_Sal )
      I_Contact( #pHs_Sal )
      Coil( "DB900_Estado_Mesas".EstadoVI[#NumeroMesaSalida].Etapa_Vacia )
   END_RUNG
   RUNG wire#w1
      I_Contact( #out_Avance_Sal )
      Contact( #pHs_Sal )
      Coil( "DB900_Estado_Mesas".EstadoVI[#NumeroMesaSalida].Etapa_Cargada )
   END_RUNG
   RUNG wire#w1
      Contact( #out_Avance_Sal )
      Coil( "DB900_Estado_Mesas".EstadoVI[#NumeroMesaSalida].Etapas_Descarga_S3 )
   END_RUNG
   // the same network as SCL:
   "DB900_Estado_Mesas".EstadoVI[#NumeroMesaSalida].Etapas_Reset := "ON" AND "DB902_Estado_ZonaMesa".EstadoMesas[#NumeroMesa].PerReset_CBx;
   "DB900_Estado_Mesas".EstadoVI[#NumeroMesaSalida].Etapa_Vacia := "ON" AND NOT #out_Avance_Sal AND NOT #pHs_Sal;
   "DB900_Estado_Mesas".EstadoVI[#NumeroMesaSalida].Etapa_Cargada := "ON" AND NOT #out_Avance_Sal AND #pHs_Sal;
   "DB900_Estado_Mesas".EstadoVI[#NumeroMesaSalida].Etapas_Descarga_S3 := "ON" AND #out_Avance_Sal;
END_REGION

REGION Network 23: ESTADOS MESA SALIDA
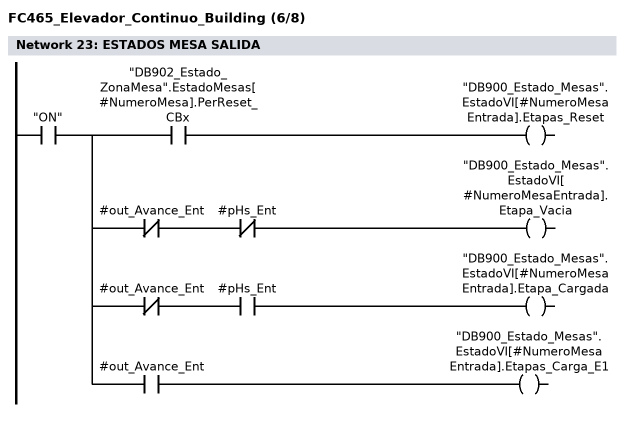
   RUNG wire#powerrail
      Contact( "ON" )
      wire#w1
      Contact( "DB902_Estado_ZonaMesa".EstadoMesas[#NumeroMesa].PerReset_CBx )
      Coil( "DB900_Estado_Mesas".EstadoVI[#NumeroMesaEntrada].Etapas_Reset )
   END_RUNG
   RUNG wire#w1
      I_Contact( #out_Avance_Ent )
      I_Contact( #pHs_Ent )
      Coil( "DB900_Estado_Mesas".EstadoVI[#NumeroMesaEntrada].Etapa_Vacia )
   END_RUNG
   RUNG wire#w1
      I_Contact( #out_Avance_Ent )
      Contact( #pHs_Ent )
      Coil( "DB900_Estado_Mesas".EstadoVI[#NumeroMesaEntrada].Etapa_Cargada )
   END_RUNG
   RUNG wire#w1
      Contact( #out_Avance_Ent )
      Coil( "DB900_Estado_Mesas".EstadoVI[#NumeroMesaEntrada].Etapas_Carga_E1 )
   END_RUNG
   // the same network as SCL:
   "DB900_Estado_Mesas".EstadoVI[#NumeroMesaEntrada].Etapas_Reset := "ON" AND "DB902_Estado_ZonaMesa".EstadoMesas[#NumeroMesa].PerReset_CBx;
   "DB900_Estado_Mesas".EstadoVI[#NumeroMesaEntrada].Etapa_Vacia := "ON" AND NOT #out_Avance_Ent AND NOT #pHs_Ent;
   "DB900_Estado_Mesas".EstadoVI[#NumeroMesaEntrada].Etapa_Cargada := "ON" AND NOT #out_Avance_Ent AND #pHs_Ent;
   "DB900_Estado_Mesas".EstadoVI[#NumeroMesaEntrada].Etapas_Carga_E1 := "ON" AND #out_Avance_Ent;
END_REGION

REGION Network 24: ESTADO MAQUINA
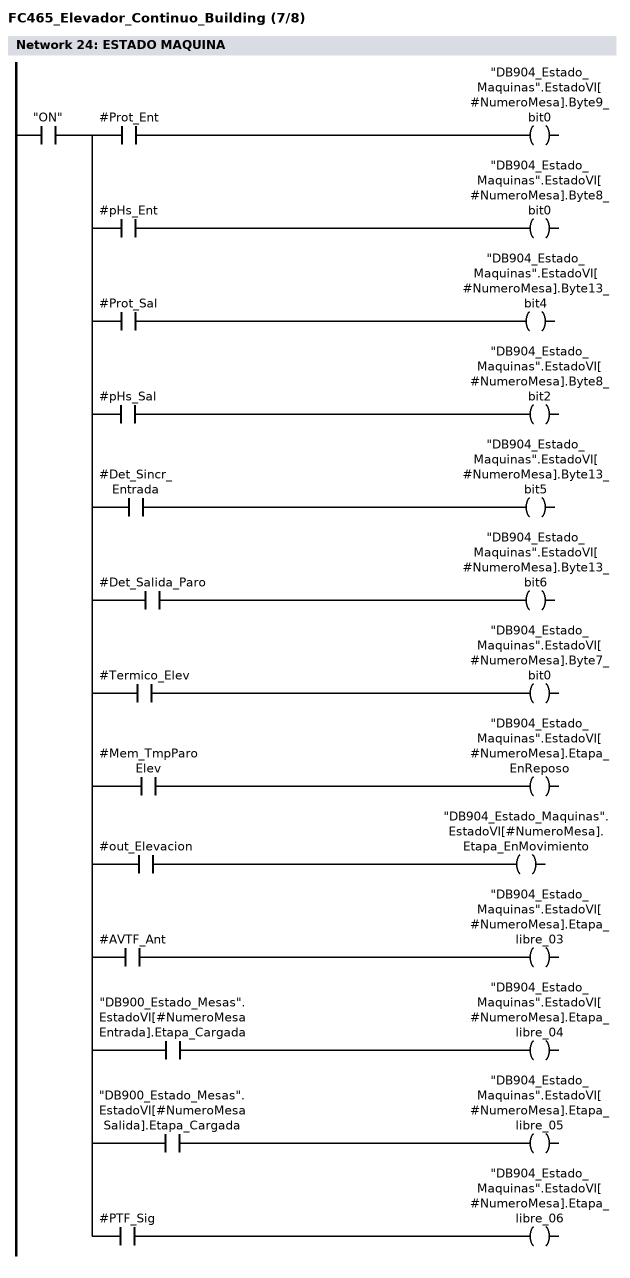
   RUNG wire#powerrail
      Contact( "ON" )
      wire#w1
      Contact( #Prot_Ent )
      Coil( "DB904_Estado_Maquinas".EstadoVI[#NumeroMesa].Byte9_bit0 )
   END_RUNG
   RUNG wire#w1
      Contact( #pHs_Ent )
      Coil( "DB904_Estado_Maquinas".EstadoVI[#NumeroMesa].Byte8_bit0 )
   END_RUNG
   RUNG wire#w1
      Contact( #Prot_Sal )
      Coil( "DB904_Estado_Maquinas".EstadoVI[#NumeroMesa].Byte13_bit4 )
   END_RUNG
   RUNG wire#w1
      Contact( #pHs_Sal )
      Coil( "DB904_Estado_Maquinas".EstadoVI[#NumeroMesa].Byte8_bit2 )
   END_RUNG
   RUNG wire#w1
      Contact( #Det_Sincr_Entrada )
      Coil( "DB904_Estado_Maquinas".EstadoVI[#NumeroMesa].Byte13_bit5 )
   END_RUNG
   RUNG wire#w1
      Contact( #Det_Salida_Paro )
      Coil( "DB904_Estado_Maquinas".EstadoVI[#NumeroMesa].Byte13_bit6 )
   END_RUNG
   RUNG wire#w1
      Contact( #Termico_Elev )
      Coil( "DB904_Estado_Maquinas".EstadoVI[#NumeroMesa].Byte7_bit0 )
   END_RUNG
   RUNG wire#w1
      Contact( #Mem_TmpParoElev )
      Coil( "DB904_Estado_Maquinas".EstadoVI[#NumeroMesa].Etapa_EnReposo )
   END_RUNG
   RUNG wire#w1
      Contact( #out_Elevacion )
      Coil( "DB904_Estado_Maquinas".EstadoVI[#NumeroMesa].Etapa_EnMovimiento )
   END_RUNG
   RUNG wire#w1
      Contact( #AVTF_Ant )
      Coil( "DB904_Estado_Maquinas".EstadoVI[#NumeroMesa].Etapa_libre_03 )
   END_RUNG
   RUNG wire#w1
      Contact( "DB900_Estado_Mesas".EstadoVI[#NumeroMesaEntrada].Etapa_Cargada )
      Coil( "DB904_Estado_Maquinas".EstadoVI[#NumeroMesa].Etapa_libre_04 )
   END_RUNG
   RUNG wire#w1
      Contact( "DB900_Estado_Mesas".EstadoVI[#NumeroMesaSalida].Etapa_Cargada )
      Coil( "DB904_Estado_Maquinas".EstadoVI[#NumeroMesa].Etapa_libre_05 )
   END_RUNG
   RUNG wire#w1
      Contact( #PTF_Sig )
      Coil( "DB904_Estado_Maquinas".EstadoVI[#NumeroMesa].Etapa_libre_06 )
   END_RUNG
   // the same network as SCL:
   "DB904_Estado_Maquinas".EstadoVI[#NumeroMesa].Byte9_bit0 := "ON" AND #Prot_Ent;
   "DB904_Estado_Maquinas".EstadoVI[#NumeroMesa].Byte8_bit0 := "ON" AND #pHs_Ent;
   "DB904_Estado_Maquinas".EstadoVI[#NumeroMesa].Byte13_bit4 := "ON" AND #Prot_Sal;
   "DB904_Estado_Maquinas".EstadoVI[#NumeroMesa].Byte8_bit2 := "ON" AND #pHs_Sal;
   "DB904_Estado_Maquinas".EstadoVI[#NumeroMesa].Byte13_bit5 := "ON" AND #Det_Sincr_Entrada;
   "DB904_Estado_Maquinas".EstadoVI[#NumeroMesa].Byte13_bit6 := "ON" AND #Det_Salida_Paro;
   "DB904_Estado_Maquinas".EstadoVI[#NumeroMesa].Byte7_bit0 := "ON" AND #Termico_Elev;
   "DB904_Estado_Maquinas".EstadoVI[#NumeroMesa].Etapa_EnReposo := "ON" AND #Mem_TmpParoElev;
   "DB904_Estado_Maquinas".EstadoVI[#NumeroMesa].Etapa_EnMovimiento := "ON" AND #out_Elevacion;
   "DB904_Estado_Maquinas".EstadoVI[#NumeroMesa].Etapa_libre_03 := "ON" AND #AVTF_Ant;
   "DB904_Estado_Maquinas".EstadoVI[#NumeroMesa].Etapa_libre_04 := "ON" AND "DB900_Estado_Mesas".EstadoVI[#NumeroMesaEntrada].Etapa_Cargada;
   "DB904_Estado_Maquinas".EstadoVI[#NumeroMesa].Etapa_libre_05 := "ON" AND "DB900_Estado_Mesas".EstadoVI[#NumeroMesaSalida].Etapa_Cargada;
   "DB904_Estado_Maquinas".EstadoVI[#NumeroMesa].Etapa_libre_06 := "ON" AND #PTF_Sig;
END_REGION

REGION Network 25: Fin de Vehiculo
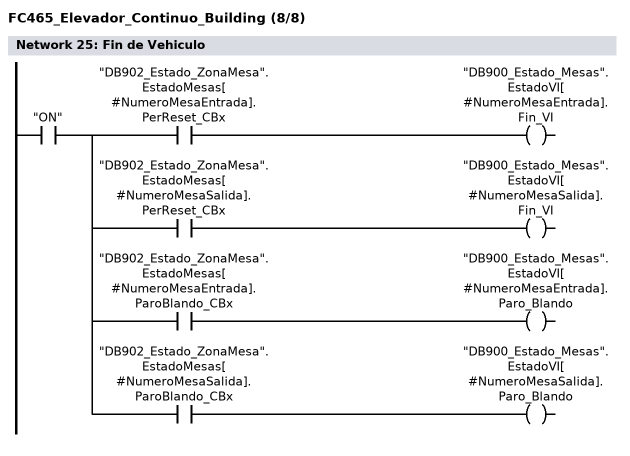
   RUNG wire#powerrail
      Contact( "ON" )
      wire#w1
      Contact( "DB902_Estado_ZonaMesa".EstadoMesas[#NumeroMesaEntrada].PerReset_CBx )
      Coil( "DB900_Estado_Mesas".EstadoVI[#NumeroMesaEntrada].Fin_VI )
   END_RUNG
   RUNG wire#w1
      Contact( "DB902_Estado_ZonaMesa".EstadoMesas[#NumeroMesaSalida].PerReset_CBx )
      Coil( "DB900_Estado_Mesas".EstadoVI[#NumeroMesaSalida].Fin_VI )
   END_RUNG
   RUNG wire#w1
      Contact( "DB902_Estado_ZonaMesa".EstadoMesas[#NumeroMesaEntrada].ParoBlando_CBx )
      Coil( "DB900_Estado_Mesas".EstadoVI[#NumeroMesaEntrada].Paro_Blando )
   END_RUNG
   RUNG wire#w1
      Contact( "DB902_Estado_ZonaMesa".EstadoMesas[#NumeroMesaSalida].ParoBlando_CBx )
      Coil( "DB900_Estado_Mesas".EstadoVI[#NumeroMesaSalida].Paro_Blando )
   END_RUNG
   // the same network as SCL:
   "DB900_Estado_Mesas".EstadoVI[#NumeroMesaEntrada].Fin_VI := "ON" AND "DB902_Estado_ZonaMesa".EstadoMesas[#NumeroMesaEntrada].PerReset_CBx;
   "DB900_Estado_Mesas".EstadoVI[#NumeroMesaSalida].Fin_VI := "ON" AND "DB902_Estado_ZonaMesa".EstadoMesas[#NumeroMesaSalida].PerReset_CBx;
   "DB900_Estado_Mesas".EstadoVI[#NumeroMesaEntrada].Paro_Blando := "ON" AND "DB902_Estado_ZonaMesa".EstadoMesas[#NumeroMesaEntrada].ParoBlando_CBx;
   "DB900_Estado_Mesas".EstadoVI[#NumeroMesaSalida].Paro_Blando := "ON" AND "DB902_Estado_ZonaMesa".EstadoMesas[#NumeroMesaSalida].ParoBlando_CBx;
END_REGION
END_FUNCTION
